FUNCTION_BLOCK PICKER_RHMI_PROXY_NEW_BA (* Communication Unit for Mirrored Picker HMI using a Socket *)
  (* Standard: 61499-2 *)
  (* Version 0.2, 2003-12-05, JHC, Rockwell Automation, Renamed from NEWCOMPFB. *)
  (* Version 0.1, 2002-01-08, JHC, Rockwell Automation, Added DLY FB as example. *)
  (* Version 0.0, 2000-05-27, JHC, Rockwell Automation *)
  (* Compiler header: package fb.rt.pnp;import fb.rt.net.*; *)
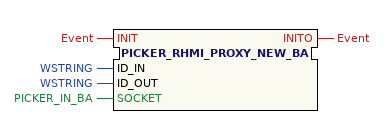
  EVENT_INPUT
    INIT; (* Initialization Request *)
  END_EVENT
  EVENT_OUTPUT
    INITO; (* Initialization Confirm *)
  END_EVENT
  VAR_INPUT
    ID_IN : WSTRING;
    ID_OUT : WSTRING;
  END_VAR
  SOCKETS
    SOCKET : PICKER_IN_BA;
  END_SOCKETS
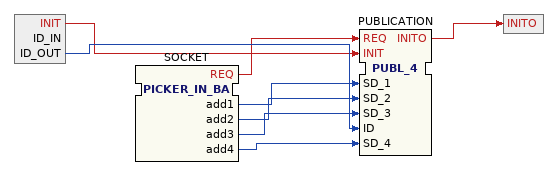
  FBS
    PUBLICATION : PUBL_4;
  END_FBS
  EVENT_CONNECTIONS
    SOCKET.REQ TO PUBLICATION.REQ;
    PUBLICATION.INITO TO INITO;
    INIT TO PUBLICATION.INIT;
  END_CONNECTIONS
  DATA_CONNECTIONS
    SOCKET.add1 TO PUBLICATION.SD_1;
    SOCKET.add2 TO PUBLICATION.SD_2;
    SOCKET.add3 TO PUBLICATION.SD_3;
    ID_OUT TO PUBLICATION.ID;
    SOCKET.add4 TO PUBLICATION.SD_4;
  END_CONNECTIONS
END_FUNCTION_BLOCK
